(* IEC 61131-3 sources: Industry-PLC-LLM/data/PLCBEAD_repo/PLCBEAD_PLCEmbed-main/PLC-BEAD/Source/GEB/METER, 1 file *)

(* ---- METER.ST ---- *)
TYPE REAL2:

	STRUCT
		R1  : REAL;
		RX : REAL;
	END_STRUCT;

END_TYPE

FUNCTION_BLOCK R2_ADD_Block

	VAR_INPUT
		X :	REAL2;
		Y :	REAL;
	END_VAR

	VAR_OUTPUT
		R2_ADD :	REAL2;
	END_VAR

	VAR
		temp :	REAL;
	END_VAR

	temp := X.RX;
	R2_ADD.RX := Y + X.R1  + X.RX;
	R2_ADD.R1  := temp - R2_ADD.RX + Y + X.R1 ;

END_FUNCTION_BLOCK

FUNCTION_BLOCK T_PLC_MS_block
	VAR_OUTPUT
		T_PLC_MS :	UDINT;
	END_VAR

	VAR
		PLC_TICKS_PER_SEC :	INT;
		PLC_SYS_TICK_CNT :	DINT;
	END_VAR

	VAR
		debug :	BOOL;(*Debug-Mode ON / OFF*)
		N :	INT;(*Debug-Faktor*)
		Offset :	UDINT;(*Debug-Offset*)
		temp :	DWORD := DWORD#1;(*Debug-Offset*)
		MODE :	BOOL;(*modus*)
		faktor :	UDINT;(*Systemtakt-Faktor*)
		init :	BOOL;
		v_plc_ticks_per_sec :	UDINT;
		base :	UDINT := UDINT#1000;
	END_VAR

	IF init = FALSE THEN
		v_plc_ticks_per_sec := INT_TO_UDINT(PLC_TICKS_PER_SEC);
		IF v_plc_ticks_per_sec = UDINT#1024 THEN
			faktor := UDINT#1;
			MODE := FALSE;
		ELSIF v_plc_ticks_per_sec > UDINT#0 THEN
			IF v_plc_ticks_per_sec <= base THEN
				faktor := base / v_plc_ticks_per_sec;
				MODE := FALSE;
			ELSE
				faktor := v_plc_ticks_per_sec / base;
				MODE := TRUE;
			END_IF;
		ELSE
			faktor := UDINT#1;
		END_IF;
		init := TRUE;
	END_IF;

	IF MODE THEN
		T_PLC_MS := DINT_TO_UDINT(PLC_SYS_TICK_CNT) / faktor;
	ELSE
		T_PLC_MS := DINT_TO_UDINT(PLC_SYS_TICK_CNT) * faktor;
	END_IF;

	IF debug THEN
		T_PLC_MS := (DWORD_TO_UDINT(SHL(UDINT_TO_DWORD(T_PLC_MS),N) OR SHL(temp,N)) - UDINT#1) + Offset;
	END_IF;
END_FUNCTION_BLOCK

FUNCTION_BLOCK METER_Block

	VAR_INPUT
		M1 :	REAL;
		M2 :	REAL;
		I1 :	BOOL;
		I2 :	BOOL;
		D :	REAL := 1.0;
		RST :	BOOL;
	END_VAR

	VAR_IN_OUT
		MX :	REAL;
	END_VAR

	VAR RETAIN
		MR :	REAL2;
	END_VAR

	VAR
		MX1 :	REAL;(*current consumPTion VALue on M1 and M2*)
		MX2 :	REAL;(*current consumPTion VALue on M1 and M2*)
		TX :	UDINT;
		last :	UDINT;
		tc :	REAL;
		init :	BOOL;
		T_PLC_MS :	T_PLC_MS_block;
		R2_ADD :	R2_ADD_Block;
	END_VAR

	T_PLC_MS();
	TX:= T_PLC_MS.T_PLC_MS;
	IF NOT init THEN
		init := TRUE;
		last := TX;
		mr.RX := mx;
		mr.R1  := 0.0;
	ELSIF TX = last THEN
		RETURN;
	ELSE
		tc := UDINT_TO_REAL(TX - last) * 0.001;
	END_IF;
	last := TX;

	(* reset *)
	IF RST THEN
		mr.R1  := 0.0;
		mr.RX := 0.0;
	ELSE
		MX1 := SEL(I1,0.0,M1);
		MX2 := SEL(I2,0.0,M2);
		R2_ADD(X:=MR,Y:=(SEL(I1,0.0,mX1) + SEL(I2, 0.0, mX2)) / D * TC);
		MR:=R2_ADD.R2_ADD;
		MX := mr.RX;
	END_IF;

END_FUNCTION_BLOCK

PROGRAM program0

	VAR
		M1 :	REAL;
		M2 :	REAL;
		I1 :	BOOL;
		I2 :	BOOL;
		D :	REAL := 1.0;
		RST :	BOOL;

		MX :	REAL;

		func_block : METER_Block;
	END_VAR

	func_block.M1 := M1;
	func_block.M2 := M2;
	func_block.I1 := I1;
	func_block.I2 := I2;
	func_block.D := D;
	func_block.RST := RST;
	func_block.MX := MX;

	func_block();

	MX  := func_block.MX;

END_PROGRAM
